INTERFACE I_ModbusTcpCore

METHOD mAddToQue : nModbusTCP_CommandStatus
VAR_INPUT
	stCommParams	: stModTcpQue;
END_VAR
END_METHOD

PROPERTY pError : BOOL
GET
END_GET
END_PROPERTY

END_INTERFACE

(* stored: Version 1.1.0.1, ProductVersion 3.1.4024.13
   Itf I_ModbusTcpCore: Id {3ca9b435-b333-4185-8859-1f049be48956}
   Method mAddToQue: Id {9d5d8193-87b3-45a1-8dee-4299bbee83fc}
   Property pError: Id {09e71c2f-a97d-48d1-bade-eb571db0b1d2}
   Get Get: Id {f46510f4-92d3-47ec-978b-2ffe0e3f0ab5} *)
